// TIA Portal V19 export
DATA_BLOCK "TokenChain"   // DB18
// stored: MemoryReserve 100
   VAR
      Data : Array[1.."TOKENCHAIN_MAX"] of "TokenChain_Data";
   END_VAR
BEGIN
   // Data[1] : CU_L1_330A1
   // Data[2] : CU_L1_340A1
   // Data[3] : CU_L1_350A1
END_DATA_BLOCK
